FUNCTION_BLOCK FB_CASE_DuplicateUpdateToDBTests EXTENDS TcUnit.FB_TestSuite

//==============================================================
//MAIN TESTS
//==============================================================

test01_();

METHOD INTERNAL test01_
VAR
	fbCase		: FB_CASE_DuplicateUpdateToDB;	
END_VAR
TcUnit.TEST('test01_');

fbCase(
	bExecute:= , 
	bUseInterimCodeForValidation:= , 
	aOCVPackStatus:= , 
	aOuterStatus:= , 
	stOCVDataDB:= , 
	stOACDataDB:= , 
	stOuterBarcodeDuplicate:= , 
	stOuterDuplicatedPackCodesFound:= , 
	stCodeInfo_Pack:= , 
	stCodeInfo_Intermediate:= , 
	stCodeInfo_Outer:= , 
	stCACData:= , 
	bDone=> , 
	bBusy=> , 
	bError=> , 
	nErrorID=> , 
	nOACFilesBlocked=> , 
	nOCVFilesBlocked=> , 
	stDaigOACDataDB=> , 
	stDiagOCVDataDB=> );

TEST_FINISHED();
END_METHOD

END_FUNCTION_BLOCK

(* stored: Version 1.1.0.1
   POU FB_CASE_DuplicateUpdateToDBTests: Id {3857eac7-9641-4b1d-9981-1db0e153c9f7}, SpecialFunc None
   Method test01_: Id {cd0bd6a3-fa13-45a2-8424-d8bddeeb9488} *)
